// TIA Portal V19 export
FUNCTION "KP8_Interface" : Void   // FC3, LAD
TITLE = Control Lights on the KP8
{ S7_Optimized_Access := 'TRUE' }
// stored: SetENOAutomatically false
   VAR_TEMP
      RetVal : Int;
      Color : Int;
      ColorStop : Int;
      ColorRun : Int;
   END_VAR
   VAR CONSTANT
      Addr : Int := 50;   // Starting Q address of the KP8
      Off : Int;   // Color
      Red : Int := 1;   // Color
      Yellow : Int := 2;   // Color
      Green : Int := 3;   // Color
      Blue : Int := 4;   // Color
      White : Int := 5;   // Color
      Switch2 : Int := 0;
      JogFwd : Int := 1;
      Stop : Int := 2;
      Reset : Int := 3;
      Switch1 : Int := 4;
      JogRev : Int := 5;
      Run : Int := 6;
      Enable : Int := 7;
   END_VAR
   VAR_TEMP   // added for the SCL form of the ladder/FBD networks
      _w1 : Bool;
      _w2 : Bool;
   END_VAR
BEGIN

REGION Network 1
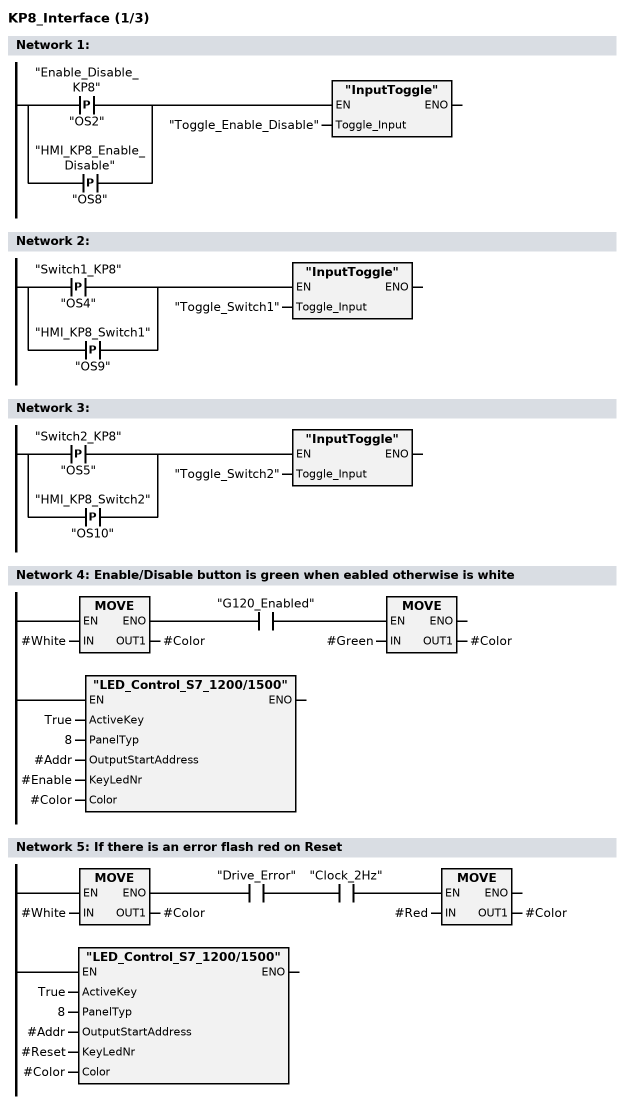
   RUNG wire#powerrail
      P_Contact(operand := "Enable_Disable_KP8", bit := "OS2")
      wire#w1
      "InputToggle"(Toggle_Input := "Toggle_Enable_Disable")
   END_RUNG
   RUNG wire#powerrail
      P_Contact(operand := "HMI_KP8_Enable_Disable", bit := "OS8")
   END_RUNG wire#w1
   // the same network as SCL:
   #_w1 := "Enable_Disable_KP8" AND NOT "OS2";   // rising edge of "Enable_Disable_KP8"
   "OS2" := "Enable_Disable_KP8";
   #_w2 := "HMI_KP8_Enable_Disable" AND NOT "OS8";   // rising edge of "HMI_KP8_Enable_Disable"
   "OS8" := "HMI_KP8_Enable_Disable";
   IF #_w1 OR #_w2 THEN "InputToggle"(Toggle_Input := "Toggle_Enable_Disable"); END_IF;
END_REGION

REGION Network 2
   RUNG wire#powerrail
      P_Contact(operand := "Switch1_KP8", bit := "OS4")
      wire#w1
      "InputToggle"(Toggle_Input := "Toggle_Switch1")
   END_RUNG
   RUNG wire#powerrail
      P_Contact(operand := "HMI_KP8_Switch1", bit := "OS9")
   END_RUNG wire#w1
   // the same network as SCL:
   #_w1 := "Switch1_KP8" AND NOT "OS4";   // rising edge of "Switch1_KP8"
   "OS4" := "Switch1_KP8";
   #_w2 := "HMI_KP8_Switch1" AND NOT "OS9";   // rising edge of "HMI_KP8_Switch1"
   "OS9" := "HMI_KP8_Switch1";
   IF #_w1 OR #_w2 THEN "InputToggle"(Toggle_Input := "Toggle_Switch1"); END_IF;
END_REGION

REGION Network 3
   RUNG wire#powerrail
      P_Contact(operand := "Switch2_KP8", bit := "OS5")
      wire#w1
      "InputToggle"(Toggle_Input := "Toggle_Switch2")
   END_RUNG
   RUNG wire#powerrail
      P_Contact(operand := "HMI_KP8_Switch2", bit := "OS10")
   END_RUNG wire#w1
   // the same network as SCL:
   #_w1 := "Switch2_KP8" AND NOT "OS5";   // rising edge of "Switch2_KP8"
   "OS5" := "Switch2_KP8";
   #_w2 := "HMI_KP8_Switch2" AND NOT "OS10";   // rising edge of "HMI_KP8_Switch2"
   "OS10" := "HMI_KP8_Switch2";
   IF #_w1 OR #_w2 THEN "InputToggle"(Toggle_Input := "Toggle_Switch2"); END_IF;
END_REGION

REGION Network 4: Enable/Disable button is green when eabled otherwise is white
   RUNG wire#powerrail
      Move(in := #White, out1 => #Color)
      Contact( "G120_Enabled" )
      Move(in := #Green, out1 => #Color)
   END_RUNG
   RUNG wire#powerrail
      "LED_Control_S7_1200/1500"(ActiveKey := True, PanelTyp := 8, OutputStartAddress := #Addr, KeyLedNr := #Enable, Color := #Color)
   END_RUNG
   // the same network as SCL:
   #Color := #White;
   IF "G120_Enabled" THEN #Color := #Green; END_IF;
   "LED_Control_S7_1200/1500"(ActiveKey := True,
                           PanelTyp := 8,
                           OutputStartAddress := #Addr,
                           KeyLedNr := #Enable,
                           Color := #Color);
END_REGION

REGION Network 5: If there is an error flash red on Reset
   RUNG wire#powerrail
      Move(in := #White, out1 => #Color)
      Contact( "Drive_Error" )
      Contact( "Clock_2Hz" )
      Move(in := #Red, out1 => #Color)
   END_RUNG
   RUNG wire#powerrail
      "LED_Control_S7_1200/1500"(ActiveKey := True, PanelTyp := 8, OutputStartAddress := #Addr, KeyLedNr := #Reset, Color := #Color)
   END_RUNG
   // the same network as SCL:
   #Color := #White;
   IF "Drive_Error" AND "Clock_2Hz" THEN #Color := #Red; END_IF;
   "LED_Control_S7_1200/1500"(ActiveKey := True,
                           PanelTyp := 8,
                           OutputStartAddress := #Addr,
                           KeyLedNr := #Reset,
                           Color := #Color);
END_REGION

REGION Network 6: Run and Stop
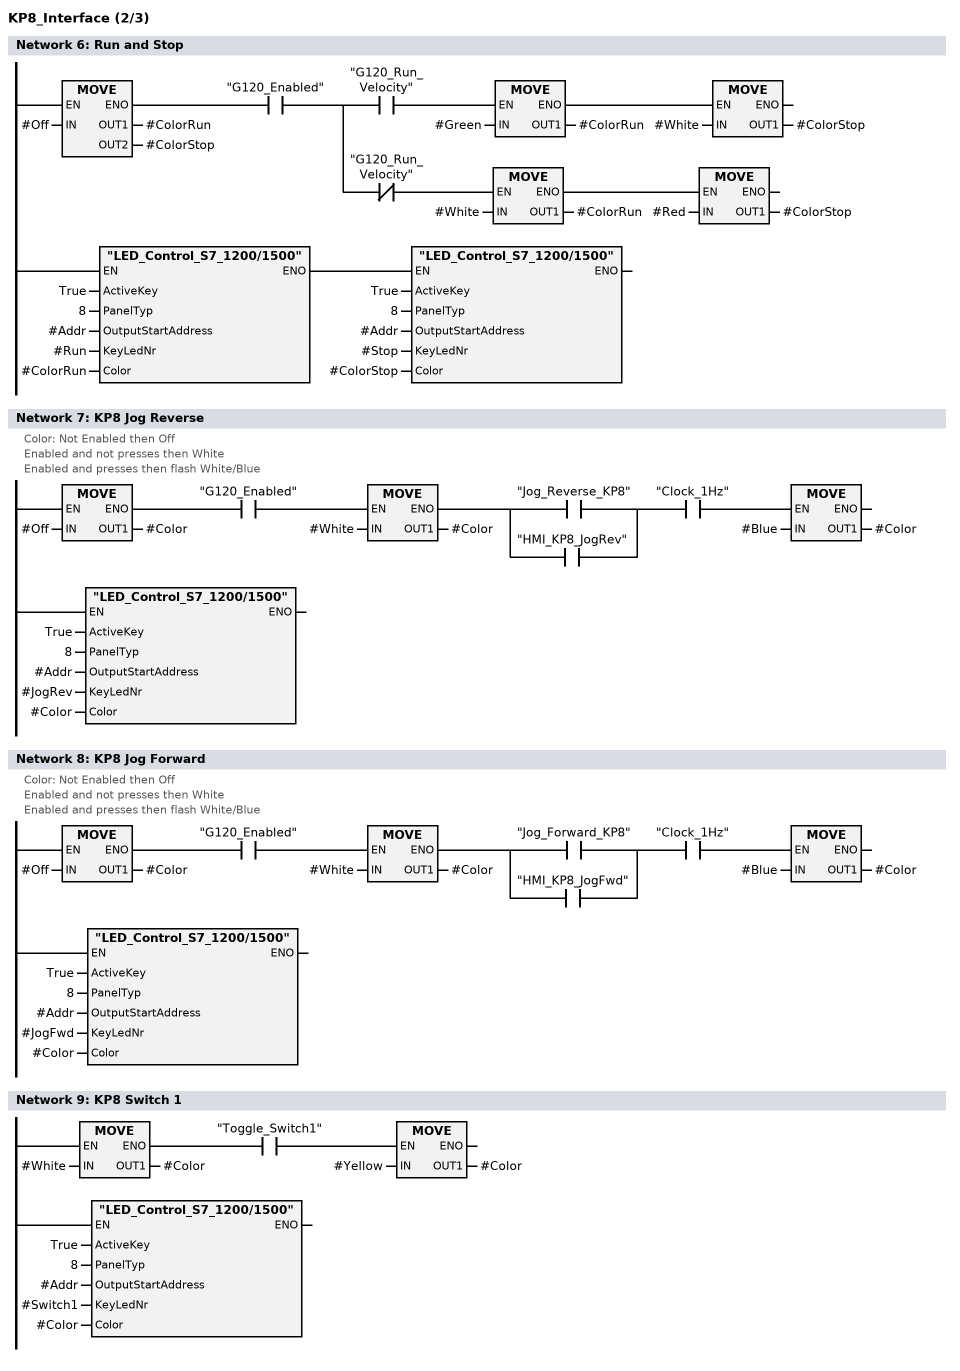
   RUNG wire#powerrail
      Move(in := #Off, out1 => #ColorRun, out2 => #ColorStop)
      Contact( "G120_Enabled" )
      wire#w1
      Contact( "G120_Run_Velocity" )
      Move(in := #Green, out1 => #ColorRun)
      Move(in := #White, out1 => #ColorStop)
   END_RUNG
   RUNG wire#w1
      I_Contact( "G120_Run_Velocity" )
      Move(in := #White, out1 => #ColorRun)
      Move(in := #Red, out1 => #ColorStop)
   END_RUNG
   RUNG wire#powerrail
      "LED_Control_S7_1200/1500"(ActiveKey := True, PanelTyp := 8, OutputStartAddress := #Addr, KeyLedNr := #Run, Color := #ColorRun)
      "LED_Control_S7_1200/1500"(ActiveKey := True, PanelTyp := 8, OutputStartAddress := #Addr, KeyLedNr := #Stop, Color := #ColorStop)
   END_RUNG
   // the same network as SCL:
   #ColorRun := #Off;
   #ColorStop := #Off;
   IF "G120_Enabled" AND "G120_Run_Velocity" THEN
       #ColorRun := #Green;
       #ColorStop := #White;
   END_IF;
   IF "G120_Enabled" AND NOT "G120_Run_Velocity" THEN
       #ColorRun := #White;
       #ColorStop := #Red;
   END_IF;
   "LED_Control_S7_1200/1500"(ActiveKey := True,
                           PanelTyp := 8,
                           OutputStartAddress := #Addr,
                           KeyLedNr := #Run,
                           Color := #ColorRun,
                           ENO => #_w1);
   IF #_w1 THEN
       "LED_Control_S7_1200/1500"(ActiveKey := True,
                               PanelTyp := 8,
                               OutputStartAddress := #Addr,
                               KeyLedNr := #Stop,
                               Color := #ColorStop);
   END_IF;
END_REGION

REGION Network 7: KP8 Jog Reverse
   // Color: Not Enabled then Off
   //             Enabled and not presses then White
   //             Enabled and presses then flash White/Blue
   RUNG wire#powerrail
      Move(in := #Off, out1 => #Color)
      Contact( "G120_Enabled" )
      Move(in := #White, out1 => #Color)
      wire#w1
      Contact( "Jog_Reverse_KP8" )
      wire#w2
      Contact( "Clock_1Hz" )
      Move(in := #Blue, out1 => #Color)
   END_RUNG
   RUNG wire#w1
      Contact( "HMI_KP8_JogRev" )
   END_RUNG wire#w2
   RUNG wire#powerrail
      "LED_Control_S7_1200/1500"(ActiveKey := True, PanelTyp := 8, OutputStartAddress := #Addr, KeyLedNr := #JogRev, Color := #Color)
   END_RUNG
   // the same network as SCL:
   #Color := #Off;
   IF "G120_Enabled" THEN #Color := #White; END_IF;
   IF "G120_Enabled" AND ("Jog_Reverse_KP8" OR "HMI_KP8_JogRev") AND "Clock_1Hz" THEN
       #Color := #Blue;
   END_IF;
   "LED_Control_S7_1200/1500"(ActiveKey := True,
                           PanelTyp := 8,
                           OutputStartAddress := #Addr,
                           KeyLedNr := #JogRev,
                           Color := #Color);
END_REGION

REGION Network 8: KP8 Jog Forward
   // Color: Not Enabled then Off
   //             Enabled and not presses then White
   //             Enabled and presses then flash White/Blue
   RUNG wire#powerrail
      Move(in := #Off, out1 => #Color)
      Contact( "G120_Enabled" )
      Move(in := #White, out1 => #Color)
      wire#w1
      Contact( "Jog_Forward_KP8" )
      wire#w2
      Contact( "Clock_1Hz" )
      Move(in := #Blue, out1 => #Color)
   END_RUNG
   RUNG wire#w1
      Contact( "HMI_KP8_JogFwd" )
   END_RUNG wire#w2
   RUNG wire#powerrail
      "LED_Control_S7_1200/1500"(ActiveKey := True, PanelTyp := 8, OutputStartAddress := #Addr, KeyLedNr := #JogFwd, Color := #Color)
   END_RUNG
   // the same network as SCL:
   #Color := #Off;
   IF "G120_Enabled" THEN #Color := #White; END_IF;
   IF "G120_Enabled" AND ("Jog_Forward_KP8" OR "HMI_KP8_JogFwd") AND "Clock_1Hz" THEN
       #Color := #Blue;
   END_IF;
   "LED_Control_S7_1200/1500"(ActiveKey := True,
                           PanelTyp := 8,
                           OutputStartAddress := #Addr,
                           KeyLedNr := #JogFwd,
                           Color := #Color);
END_REGION

REGION Network 9: KP8 Switch 1
   RUNG wire#powerrail
      Move(in := #White, out1 => #Color)
      Contact( "Toggle_Switch1" )
      Move(in := #Yellow, out1 => #Color)
   END_RUNG
   RUNG wire#powerrail
      "LED_Control_S7_1200/1500"(ActiveKey := True, PanelTyp := 8, OutputStartAddress := #Addr, KeyLedNr := #Switch1, Color := #Color)
   END_RUNG
   // the same network as SCL:
   #Color := #White;
   IF "Toggle_Switch1" THEN #Color := #Yellow; END_IF;
   "LED_Control_S7_1200/1500"(ActiveKey := True,
                           PanelTyp := 8,
                           OutputStartAddress := #Addr,
                           KeyLedNr := #Switch1,
                           Color := #Color);
END_REGION

REGION Network 10: KP8 Switch 2
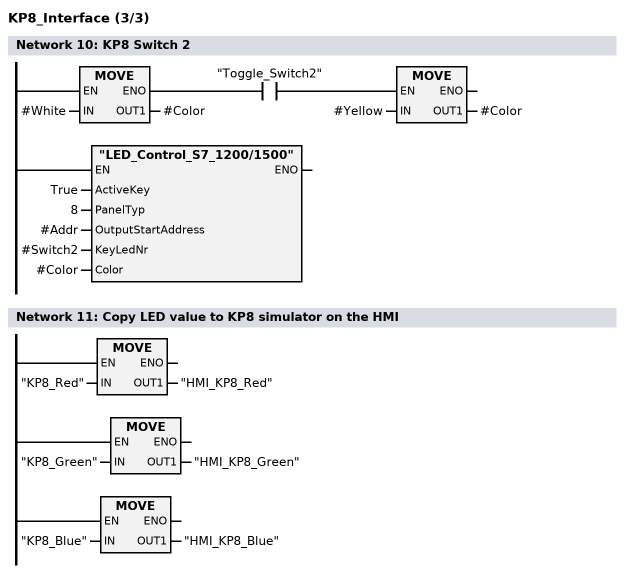
   RUNG wire#powerrail
      Move(in := #White, out1 => #Color)
      Contact( "Toggle_Switch2" )
      Move(in := #Yellow, out1 => #Color)
   END_RUNG
   RUNG wire#powerrail
      "LED_Control_S7_1200/1500"(ActiveKey := True, PanelTyp := 8, OutputStartAddress := #Addr, KeyLedNr := #Switch2, Color := #Color)
   END_RUNG
   // the same network as SCL:
   #Color := #White;
   IF "Toggle_Switch2" THEN #Color := #Yellow; END_IF;
   "LED_Control_S7_1200/1500"(ActiveKey := True,
                           PanelTyp := 8,
                           OutputStartAddress := #Addr,
                           KeyLedNr := #Switch2,
                           Color := #Color);
END_REGION

REGION Network 11: Copy LED value to KP8 simulator on the HMI
   RUNG wire#powerrail
      Move(in := "KP8_Red", out1 => "HMI_KP8_Red")
   END_RUNG
   RUNG wire#powerrail
      Move(in := "KP8_Green", out1 => "HMI_KP8_Green")
   END_RUNG
   RUNG wire#powerrail
      Move(in := "KP8_Blue", out1 => "HMI_KP8_Blue")
   END_RUNG
   // the same network as SCL:
   "HMI_KP8_Red" := "KP8_Red";
   "HMI_KP8_Green" := "KP8_Green";
   "HMI_KP8_Blue" := "KP8_Blue";
END_REGION
END_FUNCTION
